# EPICS IOC start-up script: examples/test/PSI/epp1008.iocsh
#- #############################################################################
#- mXsXXX naming
require ecmccfg v7_RC1, "NAMING=mXsXXX"

#- #############################################################################
#- add slaves
${SCRIPTEXEC} ${ecmccfg_DIR}addSlave.cmd, "HW_DESC=EPP1008, SLAVE_ID=2"

#- #############################################################################
#- apply hardware configuration
${SCRIPTEXEC} ${ecmccfg_DIR}applyConfig.cmd

#- #############################################################################
#- configure diagnostics
ecmcConfigOrDie "Cfg.EcSetDiagnostics(1)"
ecmcConfigOrDie "Cfg.EcEnablePrintouts(0)"
ecmcConfigOrDie "Cfg.EcSetDomainFailedCyclesLimit(100)"

# go active
${SCRIPTEXEC} ${ecmccfg_DIR}setAppMode.cmd
#- #############################################################################
